# EPICS autosave request: iocBoot/iocTomoStream3D_7BM/auto_settings.req
file "tomoStream.req", P=$(P), R=$(R)
file "tomoStream_settings.req", P=$(P), R=$(R)
